LIN {X 0,Y 18.289,Z 601.624,A -85,B 0,C 180,E1 -30287.78,E2 -30287.78} C_VEL
LIN {X 0,Y 13.733,Z 608.057,A -85,B 0,C 180,E1 -30330.038,E2 -30330.038} C_VEL
LIN {X 0,Y 16.56,Z 612.161,A -85,B 0,C 180,E1 -30369.58,E2 -30369.58} C_VEL
LIN {X 0,Y 24.019,Z 615.258,A -85,B 0,C 180,E1 -30391.425,E2 -30391.425} C_VEL
LIN {X 0,Y 30.034,Z 616.853,A -85,B 0,C 180,E1 -30399.441,E2 -30399.441} C_VEL
LIN {X 0,Y 31.285,Z 617.06,A -85,B 0,C 180,E1 -30403.433,E2 -30403.433} C_VEL
LIN {X 0,Y 19.66,Z 613.348,A -85,B 0,C 180,E1 -30420.002,E2 -30420.002} C_VEL
LIN {X 0,Y 13.248,Z 609.203,A -85,B 0,C 180,E1 -30452.042,E2 -30452.042} C_VEL
LIN {X 0,Y 14.264,Z 603.711,A -85,B 0,C 180,E1 -30500.222,E2 -30500.222} C_VEL
LIN {X 0,Y 21.806,Z 596.529,A -85,B 0,C 180,E1 -30528.776,E2 -30528.776} C_VEL
LIN {X 0,Y 23.813,Z 594.742,A -85,B 0,C 180,E1 -30532.573,E2 -30532.573} C_VEL
LIN {X 0,Y 24.138,Z 593.998,A -85,B 0,C 180,E1 -30535.033,E2 -30535.033} C_VEL
LIN {X 0,Y 23.36,Z 593.326,A -85,B 0,C 180,E1 -30540.433,E2 -30540.433} C_VEL
LIN {X 0,Y 21.351,Z 593.276,A -85,B 0,C 180,E1 -30548.387,E2 -30548.387} C_VEL
LIN {X 0,Y 15.562,Z 595.911,A -85,B 0,C 180,E1 -30593.775,E2 -30593.775} C_VEL
LIN {X 0,Y 17.55,Z 597.082,A -85,B 0,C 180,E1 -30619.329,E2 -30619.329} C_VEL
LIN {X 0,Y 16.258,Z 598.436,A -85,B 0,C 180,E1 -30624.107,E2 -30624.107} C_VEL
LIN {X 0,Y 7.553,Z 605.02,A -85,B 0,C 180,E1 -30662.351,E2 -30662.351} C_VEL
LIN {X 0,Y 7.434,Z 608.322,A -85,B 0,C 180,E1 -30718.29,E2 -30718.29} C_VEL
LIN {X 0,Y 15.029,Z 612.275,A -85,B 0,C 180,E1 -30759.363,E2 -30759.363} C_VEL
LIN {X 0,Y 14.765,Z 612.161,A -85,B 0,C 180,E1 -30762.287,E2 -30762.287} C_VEL
LIN {X 0,Y 5.983,Z 607.415,A -85,B 0,C 180,E1 -30808.091,E2 -30808.091} C_VEL
LIN {X 0,Y 10.28,Z 601.474,A -85,B 0,C 180,E1 -30889.934,E2 -30889.934} C_VEL
LIN {X 0,Y 20.075,Z 594.147,A -85,B 0,C 180,E1 -30908.319,E2 -30908.319} C_VEL
LIN {X 0,Y 20.405,Z 593.878,A -85,B 0,C 180,E1 -30908.656,E2 -30908.656} C_VEL
LIN {X 0,Y 19.356,Z 594.014,A -85,B 0,C 180,E1 -30913.429,E2 -30913.429} C_VEL
LIN {X 0,Y 15.927,Z 595.329,A -85,B 0,C 180,E1 -30933.813,E2 -30933.813} C_VEL
LIN {X 0,Y 15.562,Z 595.911,A -85,B 0,C 180,E1 -30953.775,E2 -30953.775} C_VEL
LIN {X 0,Y 15.185,Z 596.4,A -85,B 0,C 180,E1 -30957.89,E2 -30957.89} C_VEL
LIN {X 0,Y 13.502,Z 597.764,A -85,B 0,C 180,E1 -30961.83,E2 -30961.83} C_VEL
LIN {X 0,Y 9.445,Z 600.339,A -85,B 0,C 180,E1 -30963,E2 -30963} C_VEL
LIN {X 0,Y 5.835,Z 602.25,A -85,B 0,C 180,E1 -30954.489,E2 -30954.489} C_VEL
LIN {X 0,Y 5.091,Z 602.565,A -85,B 0,C 180,E1 -30942.075,E2 -30942.075} C_VEL
LIN {X 0,Y 5.245,Z 602.46,A -85,B 0,C 180,E1 -30938.244,E2 -30938.244} C_VEL
LIN {X 0,Y 8.942,Z 600.175,A -85,B 0,C 180,E1 -30932.227,E2 -30932.227} C_VEL
LIN {X 0,Y 9.622,Z 599.779,A -85,B 0,C 180,E1 -30948.342,E2 -30948.342} C_VEL
LIN {X 0,Y 7.027,Z 601.598,A -85,B 0,C 180,E1 -30957.166,E2 -30957.166} C_VEL
LIN {X 0,Y 5.245,Z 602.46,A -85,B 0,C 180,E1 -30938.244,E2 -30938.244} C_VEL
LIN {X 0,Y 5.245,Z 602.46,A -85,B 0,C 180,E1 -30938.244,E2 -30938.244}

QRS_NEXT_CUT()

QRS_NEXT()
QRS_HOME()

END
